FUNCTION_BLOCK FB_ReduceGantryDiff
VAR_INPUT
	xStart	:	BOOL;
END_VAR
VAR_OUTPUT
	xError	:	BOOL;
	xBusy	:	BOOL;
	xDone	:	BOOL;
END_VAR
VAR_IN_OUT
	iq_Gantry	:	HOMS_Gantry;
END_VAR
VAR
	iStep: INT;
END_VAR

(* Reduce Gantry Difference
A. Wallace, 17-3-26

On execute rising-edge, this FB decouples the gantry axes, and attempts to 
reduce the gantry difference.

Presumably the gantry error has occured due to a jammed axis.
*)

CASE iStep OF
	0: //Idle
	;
	100:
		//Decide to move P or S axis
		//Always try to move S to P if you can
		//First if the limit switches don't make sense, throw an error
		;
	//Move S
	
	//Recouple/ reset to idle
	
END_CASE

END_FUNCTION_BLOCK

(* stored: Version 1.1.0.1, ProductVersion 3.1.4024.6
   POU FB_ReduceGantryDiff: Id {5230bf37-99f3-4955-9b1e-aab6b10a65b6}, SpecialFunc None *)
